FUNCTION_BLOCK fbDatalogger_1s

VAR CONSTANT
	nRate : DINT := 1000;
	nPoints : DINT := 1000 / nRate;
END_VAR

VAR_INPUT
	fData : LREAL;
END_VAR
VAR_OUTPUT
	afLog : ARRAY[0..(nPoints-1)] OF LREAL;
	nLogJSTime : ULINT := 0;
END_VAR
VAR
	afCache : ARRAY[0..(nPoints-1)] OF LREAL;
	nCount : DINT := 0;
END_VAR

IF unixTime MOD DINT_TO_ULINT(nRate) = 0 THEN
	// Fill up the SampleArray
	afCache[nCount] := fData;
	// Increase the sampleIndex
	nCount := nCount + 1;
END_IF

IF nCount >= nPoints THEN
	// Copy values into log array
	afLog := afCache;
	// Increment log index to tell watching external logger the data has changed
	nLogJSTime := unixTime;
	// Reset count
	nCount := 0;
END_IF

END_FUNCTION_BLOCK

(* stored: Version 1.1.0.1, ProductVersion 3.1.0.36
   POU fbDatalogger_1s: Id {689e0855-648b-4318-a90d-d3c472099c5a}, SpecialFunc None *)
